# EPICS substitutions: iocBoot/iocbcur/substitutions/softMotor.substitutions
file "$(STD)/stdApp/Db/softMotor.db"
{
pattern
{SM}
{SM1}
{SM2}
{SM3}
{SM4}
{SM5}
{SM6}
{SM7}
{SM8}
{SM9}
{SM10}
{SM11}
{SM12}
{SM13}
{SM14}
{SM15}
{SM16}
}
